FUNCTION_BLOCK FB_DeadbandTester
VAR_INPUT
	fInput : LREAL;
	bEnable : BOOL;
	fConst : LREAL;
END_VAR
VAR_OUTPUT
	fOutput : LREAL;
	fXDotRef : LREAL;
END_VAR
VAR
	
END_VAR

IF bEnable THEN
	fOutput := fInput;
ELSE
	fOutput := fConst;
	fXDotRef := 0.0000001;
END_IF

END_FUNCTION_BLOCK

(* stored: Version 1.1.0.1, ProductVersion 3.1.4024.12
   POU FB_DeadbandTester: Id {f02d97ee-2672-493c-ab73-399bf476f13a}, SpecialFunc None *)
